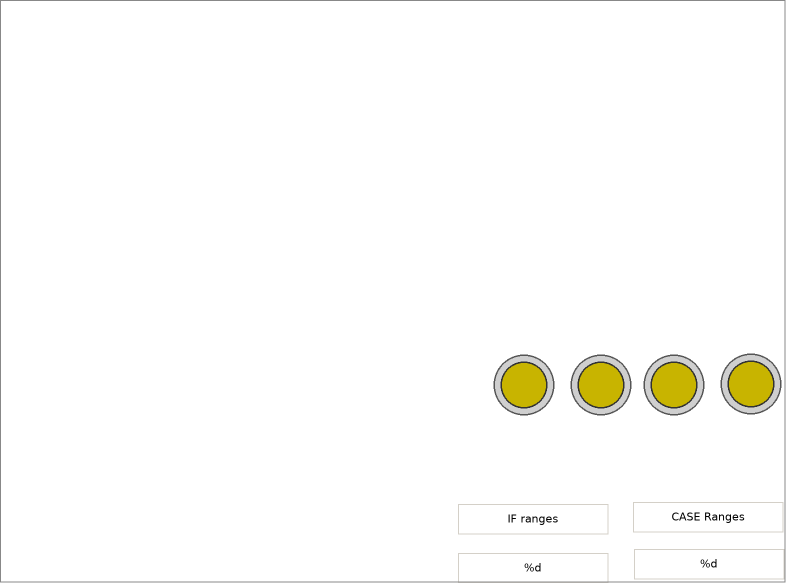
VISUALIZATION Visualization  // 786x583
    Lamp1 (489,350 70x70), variable: alights[1], style: Lamp-Lamp1-Yellow
    Textfield (458,553 150x30), "%d", text variable: NUM
        OnMouseClick: write the text variable via Edit
    Lamp1 (566,350 70x70), variable: alights[2], style: Lamp-Lamp1-Yellow
    Lamp1 (639,350 70x70), variable: alights[3], style: Lamp-Lamp1-Yellow
    Lamp1 (716,349 70x70), variable: alights[4], style: Lamp-Lamp1-Yellow
    Textfield (458,504 150x30), "IF ranges"
    Textfield (633,502 150x30), "CASE Ranges"
    Textfield (634,549 150x30), "%d", text variable: CAS
        OnMouseClick: write the text variable via Edit
END_VISUALIZATION

(* stored: Version 1.1.0.1, ProductVersion 3.1.4024.12
   Visu Visualization: Id {a12fa2e6-30f1-4a84-b0fb-f735709dc56f} *)
